DATA_BLOCK "Scanner1LoadData"
VAR
  "PLC.Station1DMXCode" : Int;
  "PLC.Station1RecipeNo" : Int;
  "PLC.PartTypeID" : String[128];
  Spare : Byte;
  "MES.ErrorCode" : Int;
  "MES.StatusBits" : DInt;
  "MES.Cycle_ID" : DInt;
  "MES.Unit_ParttypeID" : Int;
END_VAR
BEGIN
END_DATA_BLOCK
